// TwinCAT 3 PLC project PLC1
// ProgramVersion: 3.1.4023.0
// libraries:
//   Tc2_Standard, * (Beckhoff Automation GmbH)
//   Tc2_System, * (Beckhoff Automation GmbH)
//   Tc3_Module, * (Beckhoff Automation GmbH)
// project tree:
//   / PlcTask.TcTTO
//   POUs/ MAIN.TcPOU
// real-time tasks:
//   TASK PlcTask: cycle T#10ms, priority 20, ADS port 350

CONFIGURATION PLC1
    RESOURCE PLC ON TwinCAT3
        TASK PlcTask(INTERVAL := T#10ms, PRIORITY := 20);
        PROGRAM MAIN WITH PlcTask : MAIN;
    END_RESOURCE
END_CONFIGURATION

// ---- POUs/MAIN.TcPOU
PROGRAM MAIN
VAR
	intValue1 : INT;
	intValue2 : INT;
	bValue3 : BOOL;
	bValue4 : BOOL;	
	fbTON : TON;
	TEMP : BOOL:=FALSE;
END_VAR

fbTON(IN := NOT fbTON.Q, PT:= T#1S);
IF (fbTON.Q = TRUE) THEN
	IF (intValue1 <1000) THEN
		intValue1 := intValue1 +1;
		ELSE
		intValue1 :=0;		
	END_IF
	IF (intValue2 <1000) THEN
		intValue2 := intValue2 +2;
		ELSE
		intValue2 :=0;		
	END_IF
	bValue3 := NOT bValue3;
END_IF

END_PROGRAM
